# EPICS autosave request: iocBoot/ioc13Tabor/auto_settings.req
file "Tabor8024_settings.req",         P=$(P), R=$(R)
